INTERFACE I_HeatingElement EXTENDS I_ComponentBase

METHOD Off : BOOL
VAR_INPUT
END_VAR
END_METHOD

METHOD On : BOOL
VAR_INPUT
END_VAR
END_METHOD

END_INTERFACE

(* stored: Version 1.1.0.1
   Itf I_HeatingElement: Id {38dcd78f-e4ad-41ec-b17e-8151452404c0}
   Method Off: Id {aa1b184d-5420-4f86-a1e4-c0d3db7f4e1c}
   Method On: Id {ab7f4888-a4bc-4974-9946-472316fcea99} *)
